{attribute 'qualified_only'}
{attribute 'strict'}
TYPE TemperatureCompensationSources :
(
	Auto := 0, BT1, T_BT2
);
END_TYPE

(* stored: Version 1.1.0.1, ProductVersion 3.1.4024.6
   DUT TemperatureCompensationSources: Id {735a51a4-88c4-4b0d-bef4-f203a9af7fe9} *)
